{attribute 'qualified_only'}
VAR_GLOBAL
// FB DRIVE MccRev_020
	{attribute 'OPC.UA.DA' := '1'}
	bAutoButton  	   : BOOL;  // SCADA button Auto/manual Command
	{attribute 'OPC.UA.DA' := '1'}
	bForwardButton     : BOOL;  // SCADA button Forward drive Command
	{attribute 'OPC.UA.DA' := '1'}
	bReverseButton	   : BOOL;  // SCADA button Reverse drive Command
	{attribute 'OPC.UA.DA' := '1'}	 
	bTermFuse    AT%I* : BOOL;  // Term Fuse state from psyhical input
	{attribute 'OPC.UA.DA' := '1'}
	bContactor   AT%Q* : BOOL;  // Contactor state from psyhical output
	{attribute 'OPC.UA.DA' := '1'}
	udHours   		   : UDINT; // Work Time Counter - hours nonvolatile memory register
	{attribute 'OPC.UA.DA' := '1'}
	uMinutes	   	   : UINT;  // Work Time Counter - minuts nonvolatile memory register
	{attribute 'OPC.UA.DA' := '1'}
	uSeconds           : UINT;  // Work Time Counter - seconds nonvolatile memory register
	{attribute 'OPC.UA.DA' := '1'}
  	sStatus	           : T_MaxString; // Motor Status string
	{attribute 'OPC.UA.DA' := '1'}
	sState 	           : T_MaxString; // Motor State string		

END_VAR

(* stored: Version 1.1.0.1, ProductVersion 3.1.4024.12
   GVL MccRev_020: Id {35b2ef9f-0d01-42d9-8216-8626b79eeddc} *)
